TYPE
    ST_Auto_Allocated :
    STRUCT
    END_STRUCT
END_TYPE

(* stored: Version 1.1.0.1, ProductVersion 3.1.4024.13
   DUT ST_Auto_Allocated: Id {0f921436-3bf2-4938-922a-eb5ddc4fe8c2} *)
